// SIMATIC S7-200 SMART project (STEP 7-Micro/WIN SMART), CPU SR40

SYMBOL_TABLE 表格 1
过程变量             VW0
PID输出            VW2
手动输入             VD4
设定值              VD8
YLAST1           VD100
YLAST2           VD104
YLAST3           VD108
END_SYMBOL_TABLE

SYMBOL_TABLE 系统符号
Always_On        SM0.0    // 始终接通
First_Scan_On    SM0.1    // 仅在第一个扫描周期时接通
Clock_1s         SM0.5    // 针对 1 s 的周期时间，时钟脉冲接通 0.5 s，断开 0.5 s。
Time_1_Intrvl    SMB35    // 指定中断 1 的时间间隔（从 1 - 255，以 1 ms 递增）。
END_SYMBOL_TABLE

ORGANIZATION_BLOCK MAIN:OB1
TITLE=程序注释
BEGIN
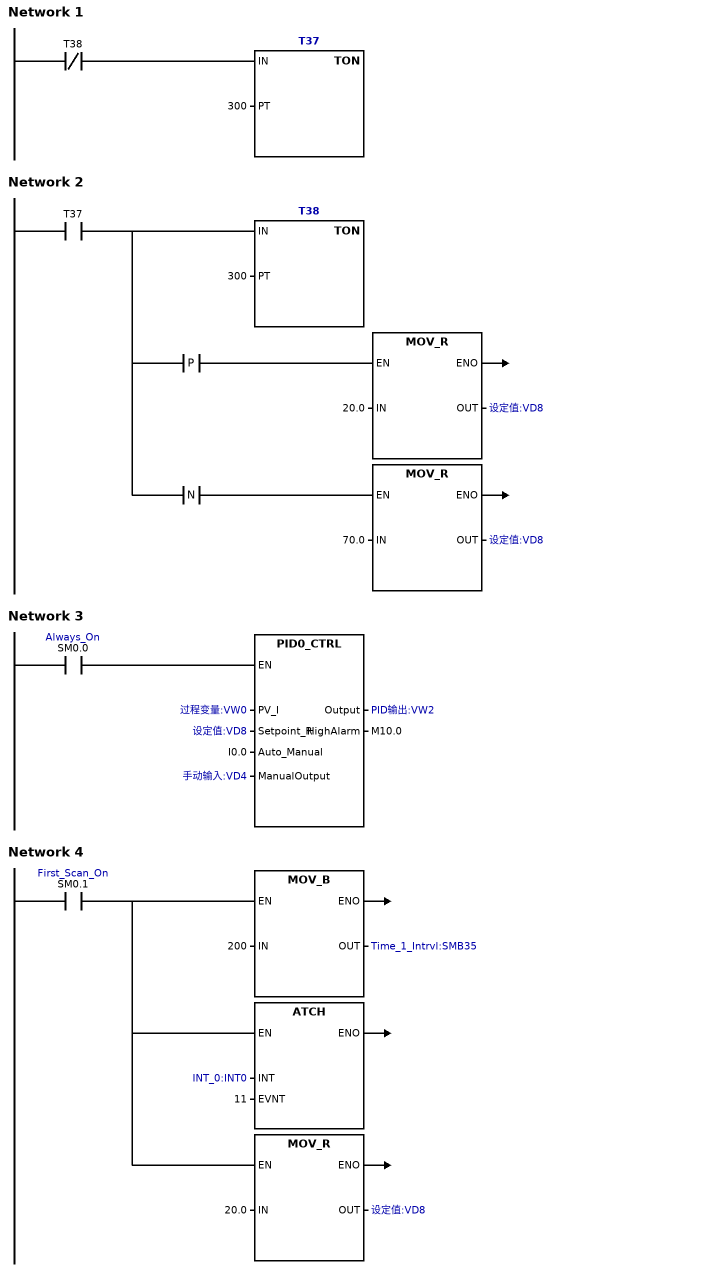
Network 1
LDN    T38
TON    T37, 300
Network 2
LD     T37
LPS
TON    T38, 300
EU
MOVR   20.0, 设定值:VD8
LPP
ED
MOVR   70.0, 设定值:VD8
Network 3
LD     Always_On:SM0.0
CALL   PID0_CTRL:SBR1, 过程变量:VW0, 设定值:VD8, I0.0, 手动输入:VD4, PID输出:VW2, M10.0
Network 4
LD     First_Scan_On:SM0.1
MOVB   200, Time_1_Intrvl:SMB35
ATCH   INT_0:INT0, 11
MOVR   20.0, 设定值:VD8
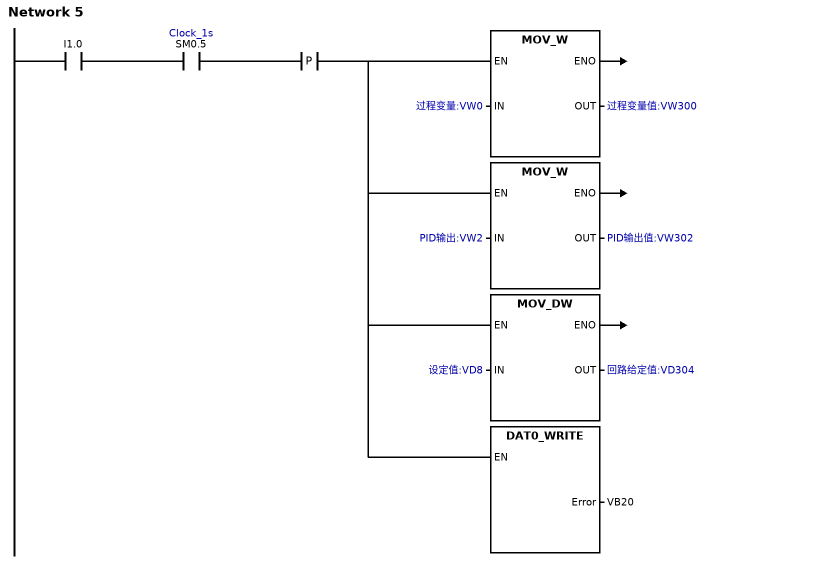
Network 5
//SM0.5产生周期为1s的时钟脉冲
//上升沿检测
//过程变量值送数据日志缓冲区
//PID输出值送数据日志缓冲区
//回路设定值送数据日志缓冲区
//保存缓冲区中的数据
LD     I1.0
A      Clock_1s:SM0.5
EU
MOVW   过程变量:VW0, 过程变量值:VW300
MOVW   PID输出:VW2, PID输出值:VW302
MOVD   设定值:VD8, 回路给定值:VD304
CALL   DAT0_WRITE:SBR2, VB20
END_ORGANIZATION_BLOCK

// SBR0: protected block, not included

// SBR1: protected block, not included

// SBR2: protected block, not included

INTERRUPT_BLOCK INT_0:INT0
TITLE=中断例程注释
BEGIN
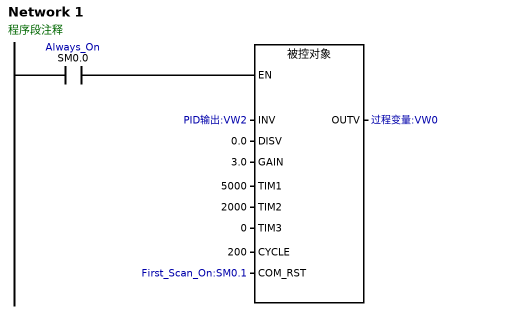
Network 1
// 程序段注释
LD     Always_On:SM0.0
CALL   被控对象:SBR0, PID输出:VW2, 0.0, 3.0, 5000, 2000, 0, 200, First_Scan_On:SM0.1, 过程变量:VW0
END_INTERRUPT_BLOCK

// INT1: protected block, not included
